(* IEC 61131-3 sources: repolevel_ST_code_completion/output/0121完整版本/repoeval_counter/readful_result_no_provide, 1 file *)

(* ---- FB_counter.st ---- *)
VAR
    nPrevValue: INT;   (* Previous value for internal tracking *)
END_VAR

IF bReset THEN
    nValue := 0;       (* Reset the counter *)
ELSIF bUp THEN
    nValue := nValue + 1; (* Increment the counter *)
ELSIF bDown THEN
    nValue := nValue - 1; (* Decrement the counter *)
END_IF
END_FUNCTION_BLOCK
